FUNCTION CheckDivDWord : DWORD
VAR_INPUT
	divisor				: DWORD;
END_VAR
VAR
END_VAR

IF divisor = 0 THEN
	CheckDWordZeroDiv_ErrCnt := CheckDWordZeroDiv_ErrCnt + 1;
	CheckDivDWord := 1;
ELSE
	CheckDivDWord := divisor;
END_IF

END_FUNCTION

(* stored: Version 1.1.0.1, ProductVersion 3.1.4024.9
   POU CheckDivDWord: Id {7ce57a42-f5a6-44da-b65b-7083a108e1cb}, SpecialFunc CheckDivInt64 *)
